// TIA Portal V18 export
ORGANIZATION_BLOCK "Main"   // OB1, LAD, ProgramCycle
TITLE = "Main Program Sweep (Cycle)"
{ S7_Optimized_Access := 'TRUE' }
// stored: SetENOAutomatically false
   VAR_INPUT
      Initial_Call : Bool;   // Initial call of this OB
      Remanence : Bool;   // =True, if remanent data are available
   END_VAR
BEGIN

REGION Network 1: Test comment
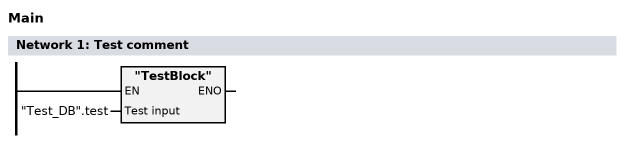
   RUNG wire#powerrail
      "TestBlock"("Test input" := "Test_DB".test)
   END_RUNG
   // the same network as SCL:
   "TestBlock"("Test input" := "Test_DB".test);
END_REGION
END_ORGANIZATION_BLOCK
